(* IEC 61131-3 sources: repolevel_ST_code_completion/output/0127完整版本_带planner/repoeval_elevator/readful_result_history, 5 files *)

(* ---- F_DetectCurrentFloor_0.st ---- *)
FUNCTION F_DetectCurrentFloor : INT
VAR_INPUT
	FloorSensor0	:	BOOL;		// 0楼传感器
	FloorSensor1	:	BOOL;		// 1楼传感器
	FloorSensor2	:	BOOL;		// 2楼传感器
	FloorSensor3	:	BOOL;		// 3楼传感器
	CurrentFloor	:	INT;		// 当前楼层（用于保持状态）
END_VAR
IF FloorSensor0 THEN
	F_DetectCurrentFloor := 0;
ELSIF FloorSensor1 THEN
	F_DetectCurrentFloor := 1;
ELSIF FloorSensor2 THEN
	F_DetectCurrentFloor := 2;
ELSIF FloorSensor3 THEN
	F_DetectCurrentFloor := 3;
ELSE
	F_DetectCurrentFloor := CurrentFloor;
END_IF;
RETURN;
END_FUNCTION

(* ---- F_RegisterCalls_0.st ---- *)
FUNCTION F_RegisterCalls
VAR_INPUT
	CallGround		:	BOOL;		// 0楼呼叫
	CallFloor1		:	BOOL;		// 1楼呼叫
	CallFloor2		:	BOOL;		// 2楼呼叫
	CallFloor3		:	BOOL;		// 3楼呼叫
END_VAR
VAR_IN_OUT
	TargetFloors	:	ARRAY[0..3] OF BOOL;	// 目标楼层数组
END_VAR
IF CallGround THEN
	TargetFloors[0] := TRUE;
END_IF

IF CallFloor1 THEN
	TargetFloors[1] := TRUE;
END_IF

IF CallFloor2 THEN
	TargetFloors[2] := TRUE;
END_IF

IF CallFloor3 THEN
	TargetFloors[3] := TRUE;
END_IF

RETURN;
END_FUNCTION

(* ---- F_UpdateDoorAnimation_0.st ---- *)
FUNCTION F_UpdateDoorAnimation : DINT
VAR_INPUT
	bOpenDoor		:	BOOL;		// 开门命令
	bCloseDoor		:	BOOL;		// 关门命令
	bCallFloor		:	BOOL;		// 该楼层有呼叫
	nCurrentAni		:	DINT;		// 当前动画值
	nMaxAni			:	DINT := 70;	// 最大动画值
END_VAR
VAR
	nNewAni			:	DINT;		// 新的动画值
END_VAR

nNewAni := nCurrentAni;

// 开门动画（增加动画值）
IF bOpenDoor AND nNewAni < nMaxAni THEN
	nNewAni := nNewAni + 1;
END_IF

// 关门动画（减少动画值）
IF bCloseDoor AND nNewAni > 0 THEN
	nNewAni := nNewAni - 1;
END_IF

// 楼层呼叫动画（增加动画值）
IF bCallFloor AND nNewAni < nMaxAni THEN
	nNewAni := nNewAni + 1;
END_IF

// 保持动画值不变
IF NOT bCallFloor AND NOT bOpenDoor AND NOT bCloseDoor THEN
	nNewAni := nCurrentAni;
END_IF

F_UpdateDoorAnimation := nNewAni;
END_FUNCTION

(* ---- FB_ElevatorDoorController_0.st ---- *)
FUNCTION_BLOCK FB_ElevatorDoorController
VAR_INPUT
	bArrivedAtTarget	:	BOOL;		// 到达目标楼层
	bDoorClosed			:	BOOL;		// 门已关闭传感器
END_VAR
VAR_OUTPUT
	bOpenDoor			:	BOOL;		// 开门命令
	bCloseDoor			:	BOOL;		// 关门命令
	bDoorOpen			:	BOOL;		// 门打开状态
	bDoorReady			:	BOOL;		// 门准备好（可以移动）
END_VAR
VAR
	fbDoorTimer			:	TON;		// 开门延时定时器
	fbCloseDoorTimer	:	TON;		// 关门延时定时器
	nState				:	INT;		// 状态机
	bEmergencyStop		:	BOOL;		// 紧急停止信号
END_VAR

CASE nState OF
	0: // 空闲状态
		bOpenDoor := FALSE;
		bCloseDoor := FALSE;
		bDoorOpen := FALSE;
		bDoorReady := TRUE;

		IF bArrivedAtTarget THEN
			nState := 1; // 开始开门流程
		END_IF

	1: // 开门延时
		bCloseDoor := FALSE;
		bDoorReady := FALSE;
		bOpenDoor := TRUE;
		fbDoorTimer(IN := TRUE, PT := T#2S);

		IF fbDoorTimer.Q THEN
			fbDoorTimer(IN := FALSE);
			nState := 2; // 门打开状态
		END_IF

	2: // 门打开状态
		bDoorOpen := TRUE;
		bOpenDoor := FALSE;

		IF NOT bArrivedAtTarget THEN
			nState := 3; // 开始关门流程
		END_IF

	3: // 关门延时
		bOpenDoor := FALSE;
		bDoorOpen := FALSE;
		bCloseDoor := TRUE;
		fbCloseDoorTimer(IN := TRUE, PT := T#2S);

		IF fbCloseDoorTimer.Q THEN
			fbCloseDoorTimer(IN := FALSE);
			nState := 4; // 检查门关闭状态
		END_IF

	4: // 检查门关闭状态
		bCloseDoor := FALSE;

		IF bDoorClosed THEN
			bDoorReady := TRUE;
			nState := 0; // 返回空闲状态
		END_IF

ELSE
	// 异常处理
	bOpenDoor := FALSE;
	bCloseDoor := FALSE;
	bDoorOpen := FALSE;
	bDoorReady := FALSE;
	nState := 0; // 返回空闲状态
END_CASE
END_FUNCTION_BLOCK

(* ---- FB_ElevatorMovement_0.st ---- *)
FUNCTION_BLOCK FB_ElevatorMovement
VAR_INPUT
	CurrentFloor		:	INT;				// 当前楼层
	bDoorReady			:	BOOL;				// 门准备好
END_VAR
VAR_IN_OUT
	TargetFloors		:	ARRAY[0..3] OF BOOL;	// 目标楼层数组
END_VAR
VAR_OUTPUT
	bMovingUp			:	BOOL;				// 向上移动
	bMovingDown			:	BOOL;				// 向下移动
	bArrivedAtTarget	:	BOOL;				// 到达目标楼层
END_VAR
VAR
	i					:	INT;				// 循环变量
	bHasUpperRequest	:	BOOL;				// 有更高楼层请求
	bHasLowerRequest	:	BOOL;				// 有更低楼层请求
END_VAR

// 初始化状态变量
bHasUpperRequest := FALSE;
bHasLowerRequest := FALSE;

// 遍历目标楼层数组
FOR i := 0 TO 3 DO
	IF TargetFloors[i] THEN
		IF (i > CurrentFloor) AND bDoorReady THEN
			bHasUpperRequest := TRUE;
		ELSIF (i < CurrentFloor) AND bDoorReady THEN
			bHasLowerRequest := TRUE;
		END_IF;
	END_IF;
END_FOR

// 根据请求状态设置移动方向
IF bHasUpperRequest THEN
	bMovingUp := TRUE;
	bMovingDown := FALSE;
ELSIF bHasLowerRequest THEN
	bMovingDown := TRUE;
	bMovingUp := FALSE;
ELSE
	bMovingUp := FALSE;
	bMovingDown := FALSE;
END_IF

// 检查是否到达目标楼层
IF TargetFloors[CurrentFloor] THEN
	IF bDoorReady THEN
		bArrivedAtTarget := TRUE;
		TargetFloors[CurrentFloor] := FALSE; // 清除请求
		bMovingUp := FALSE;
		bMovingDown := FALSE;
	ELSE
		bArrivedAtTarget := FALSE;
	END_IF;
ELSE
	bArrivedAtTarget := FALSE;
END_IF
END_FUNCTION_BLOCK
